Staubli VAL3: DialogOKandBI.pgx

public program dialogOKandBI(dio x_diBreakInput, string x_sTitle, string x_sText_r1, string x_sText_r2, string x_sText_r3, string x_sText_r4)
  local num l_nNum
begin

  //notes: screen size is 13rowsX40columns
 //usage: call DialogOnlyBI(diStartButton, "START PROGRAM", "Press Start Button or F1", "to start the program", "", "", sUserScreen)

  wait(getKey()==-1)
  userPage()
  call clrscr()

  call sCenterTitle(x_sTitle)

  title(x_sTitle)

  gotoxy(0,4)
  call sCenterRow(x_sText_r1)
  putln(x_sText_r1)

  gotoxy(0,5)
  call sCenterRow(x_sText_r2)
  putln(x_sText_r2)

  gotoxy(0,6)
  call sCenterRow(x_sText_r3)
  putln(x_sText_r3)

  gotoxy(0,7)
  call sCenterRow(x_sText_r4)
  putln(x_sText_r4)

  gotoxy(0,13)
  put("F1=Ok")

  getKey()
  do
    l_nNum=getKey()
    delay(0)
  until l_nNum==271 or x_diBreakInput==true

  call clrscr()
  wait(getKey()==-1)

end
